// TIA Portal V19 export
FUNCTION "PPrg_Call" : Void   // FC7, LAD
// stored: SetENOAutomatically false
BEGIN
END_FUNCTION
